PROGRAM MAIN
VAR
END_VAR

END_PROGRAM

(* stored: Version 1.1.0.1
   POU MAIN: Id {a256f1ed-2fdb-47cd-bbe2-4ea5cda6d818} *)
